(* IEC 61131-3 sources: Industry-PLC-LLM/data/PLCBEAD_repo/PLCBEAD_PLCEmbed-main/PLC-BEAD/Source/GEB/INC1, 1 file *)

(* ---- INC1.ST ---- *)
FUNCTION INC1:INT

	VAR_INPUT
		X :	INT;
		N :	INT;
	END_VAR

	IF X >= N - 1 THEN
		INC1 := 0;
	ELSE
		INC1 := X + 1;
	END_IF;
END_FUNCTION

PROGRAM program0
  VAR
	X :	INT;
	N :	INT;
    CEIL5_OUT : INT;
  END_VAR

  CEIL5_OUT := INC1(X, N);
END_PROGRAM
